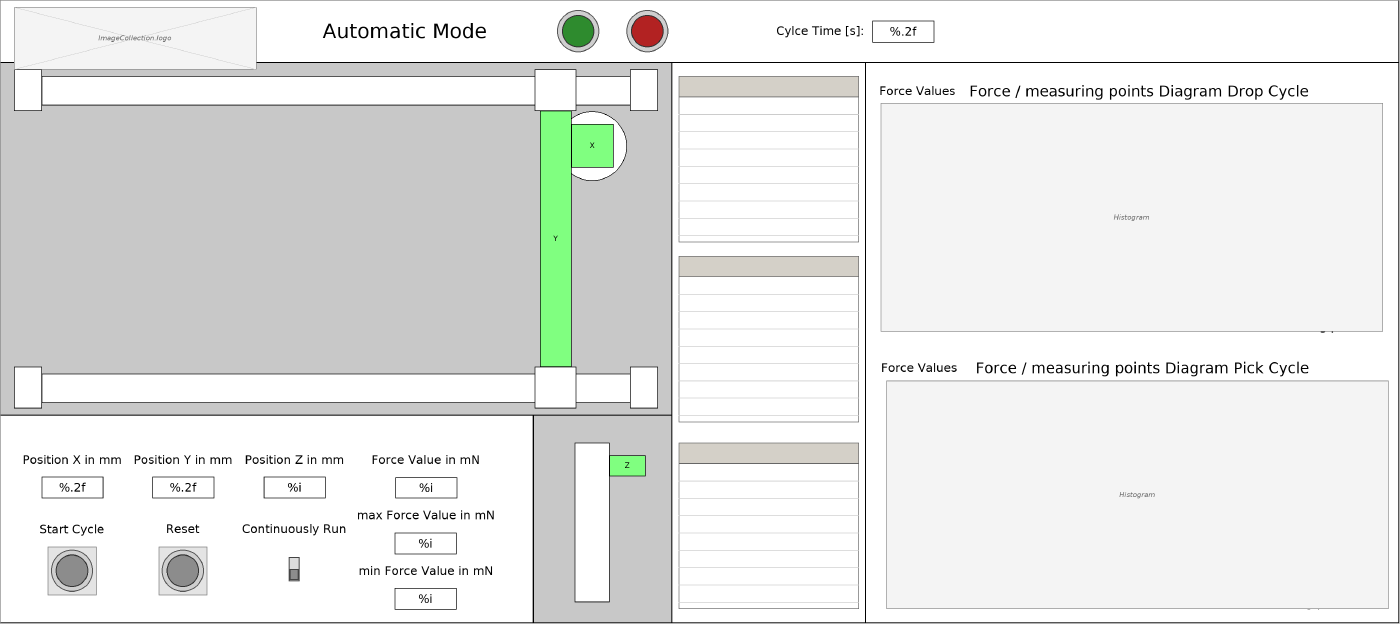
VISUALIZATION AutomaticMode  // 2022x902
    Rectangle (1250,90 770x810)
    Rectangle (0,600 770x300)
    Rectangle (970,90 280x810)
    Rectangle (0,0 2020x90)
    Rectangle (770,600 200x300)
    Rectangle (0,90 970x510)
    Ellipse (805,161 100x100)
        p3528305787: realVisuDiskY
        p2773130477: realVisuDiskX
        p874137650: realVisuDiskY
        p1126004900: realVisuDiskX
    Rectangle (60,110 852x42)
    Rectangle (60,540 852x42)
    PushSwitch (69,790 70x70), variable: MAIN.bStart, behaviour: TAP, style: Switch-PushSwitch-Gray
    Label (54,750 100x30), "Start Cycle"
    PushSwitch (229,790 70x70), variable: bReset, behaviour: TAP, style: Switch-PushSwitch-Gray
    Label (229,750 70x29), "Reset"
    Rectangle (825,179 61x63), "X", colour toggle: setError.Q1
        p3560616238: realVisuPosY
        p2738717112: realVisuPosX
    DipSwitch (390,805 70x35), variable: MAIN.bDauerlauf, behaviour: TOGGLE, style: Switch-DipSwitch-Gray
    Label (350,750 150x29), "Continuously Run"
    Rectangle (60,689 89x31), "%.2f", text variable: posAxisX.Position
    Label (30,650 149x29), "Position X in mm"
    Rectangle (220,689 89x31), "%.2f", text variable: posAxisY.Position
    Label (190,650 149x29), "Position Y in mm"
    Lamp1 (800,10 70x70), variable: NOT bEmergencyPressed AND NOT globalErrorDetect, style: Lamp-Lamp1-green
    Lamp1 (900,10 70x70), variable: bEmergencyPressed OR globalErrorDetect, style: Lamp-Lamp1-Red
    Rectangle (880,658 52x30), "Z", colour toggle: setError.Q1
        p2738717112: intVisuPosZ
    Rectangle (830,640 50x230)
    Rectangle (381,689 89x31), "%i", text variable: posAxisZ
    Label (351,650 149x29), "Position Z in mm"
    Rectangle (571,690 89x30), "%i", text variable: acutalForceValue
    Label (530,650 170x29), "Force Value in mN"
    Rectangle (570,770 89x31), "%i", text variable: maxForceValuePos
    Label (510,730 210x29), "max Force Value in mN"
    Rectangle (570,850 89x31), "%i", text variable: maxForceValueNeg
    Label (510,810 210x30), "min Force Value in mN"
    Label (460,20 250x50), "Automatic Mode"
    Group (1270,110 727x383)
        Label (120,0 510x44), "Force / measuring points Diagram Drop Cycle"
        Label (550,340 160x43), "measuring points"
        Label (0,0 110x43), "Force Values"
        Histogram (2,39 725x330), scale format: %.1f, scale -10000..3000
            p518627256: mN
            p1518820177: visu.forceMemoryDrop.sArrForceValue
            p102497268: visu.forceMemoryDrop.sArrForceValue
            p788070771: ARRAY [BufStart..BufEnd] OF INT
    Table (980,370 260x240), data array: visu.stringErrorText
        p3854506369: visu.stringErrorText[INDEX]
        p2232123230: Error Messages
    Table (980,110 260x240), data array: visu.stringMessageText
        p3854506369: visu.stringMessageText[INDEX]
        p2232123230: Status Messages
    Table (980,640 260x240), data array: visu.stringDebugText
        p3854506369: visu.stringDebugText[INDEX]
        p2232123230: Debug Messages
    Group (1270,510 735x383)
        Label (530,340 160x43), "measuring points"
        Label (120,0 520x44), "Force / measuring points Diagram Pick Cycle"
        Label (0,0 115x43), "Force Values"
        Histogram (10,40 725x330), scale format: %.1f, scale -3000..13000
            p518627256: mN
            p1518820177: visu.forceMemoryPick.sArrForceValue
            p102497268: visu.forceMemoryPick.sArrForceValue
            p788070771: ARRAY [BufStart..BufEnd] OF INT
    Rectangle (780,160 45x370), "Y", colour toggle: setError.Q1
        p3560616238: realVisuPosY
    Rectangle (772,100 60x60)
        p3560616238: realVisuPosY
    Rectangle (772,530 60x60)
        p3560616238: realVisuPosY
    Rectangle (20,100 40x60)
    Rectangle (910,100 40x60)
    Rectangle (20,530 40x60)
    Rectangle (910,530 40x60)
    Image (20,10 350x90), image: ImageCollection.logo
    Rectangle (1260,30 89x31), "%.2f", text variable: visu.TimeDifSec
    Label (1110,30 149x29), "Cylce Time [s]:"
END_VISUALIZATION

(* stored: Version 1.1.0.1, ProductVersion 3.1.4018.2
   Visu AutomaticMode: Id {eb9e94f6-82bd-474b-bb24-ea6f6e100d51} *)
